SYSTEM System (* System Configuration *)
  (* Version 0.0, 10/1/2026, Schneider Electric *)
  APPLICATION APP1
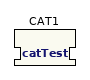
    FBS
      CAT1 : catTest;
    END_FBS
  END_APPLICATION
  DEVICE EcoRT_0 : Soft_dPAC
    RESOURCE RES0 : EMB_RES_ECO
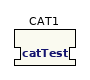
      FBS
        CAT1 : catTest;
      END_FBS
    END_RESOURCE
  END_DEVICE
  MAPPINGS
    APP1.CAT1 ON EcoRT_0.RES0;
  END_MAPPINGS
END_SYSTEM
(* other elements stored in the file *)
(* DefaultLayer Name=Default *)
